{attribute 'enable_dynamic_creation'}
{attribute 'no_assign'}
FUNCTION_BLOCK FB_Stack EXTENDS FB_Collection IMPLEMENTS I_Stack
VAR_INPUT
	ipList : I_List; // List to perform operations on.
END_VAR
VAR_OUTPUT
END_VAR

(* Number of elements in the stack *)
PROPERTY _Count : T_Capacity
GET
IF THIS^.NullReferenceException() THEN _Count := -1; RETURN; END_IF
_Count := THIS^.ipList._Count;
END_GET
END_PROPERTY

PROPERTY _Error_Status : ST_ERROR
GET
IF THIS^.NullReferenceException() THEN _Error_Status := THIS^.stError; RETURN; END_IF
THIS^.stError := THIS^.ipList._Error_Status;
_Error_Status := F_Error(THIS^.stError.bSTATUS, THIS^.stError.nCODE, THIS^.stError.sSOURCE);
END_GET
END_PROPERTY

(* Checks of stack is empty.*)
PROPERTY _Is_Empty : BOOL
GET
IF THIS^.NullReferenceException() THEN _Is_Empty := TRUE; RETURN; END_IF
_Is_Empty := THIS^.ipList._Is_Empty;
END_GET
END_PROPERTY

METHOD PROTECTED CatchError : BOOL
VAR_INPUT
END_VAR
stError := THIS^.ipList._Error_Status;
CatchError := stError.bSTATUS;
END_METHOD

(* Empties/Clears/Deletes every item on the stack*)
METHOD Clear
VAR_INPUT
END_VAR
IF THIS^.NullReferenceException() THEN RETURN; END_IF
THIS^.ipList.Clear();
END_METHOD

METHOD PROTECTED NullReferenceException : BOOL
NullReferenceException := THIS^.ipList = 0;
IF NOT NullReferenceException THEN RETURN; END_IF
THIS^.RaiseException(2000+GVL_CmpErrors.ERR_INVALID_REFERENCE, 'Null or Invalid Reference');
END_METHOD

(* Get item from stack without removing it. *)
METHOD Peek : I_Stack
VAR_INPUT
	Item 	: ANY; (* Variable to store returned item value *)
	nIndex 	: DINT; (* Location of item*)
END_VAR
VAR_OUTPUT
	bSuccess : BOOL;
END_VAR
Peek := THIS^;
IF THIS^.NullReferenceException() THEN RETURN; END_IF
THIS^.ipList.Get(Item, nIndex, bSuccess => bSuccess);
END_METHOD

(* Gets and deletes item at the top of the stack *)
METHOD Pop : I_Stack
VAR_INPUT
	Item : ANY; (* Variable to store returned item value *)
END_VAR
VAR_OUTPUT
	bSuccess : BOOL;
END_VAR
VAR
	bA, bB 	 : BOOL;
END_VAR
Pop := THIS^;
IF THIS^.NullReferenceException() THEN RETURN; END_IF
THIS^.ipList.Get_First(Item, bSuccess => bA).Remove( bSuccess => bB);
bSuccess := bA AND bB;
END_METHOD

(* Removes item at the top of the stack without returning anything *)
METHOD Pop_Void : I_Stack
VAR_OUTPUT
	bSuccess : BOOL;
END_VAR
Pop_Void := THIS^;
IF THIS^.NullReferenceException() THEN RETURN; END_IF
THIS^.ipList.Remove(bSuccess => bSuccess);
END_METHOD

(* Add item to the top of the stack *)
METHOD Push : I_Stack
VAR_INPUT
	Item : ANY; (* Variable containg data to store on the stack *)
END_VAR
VAR_OUTPUT
	bSuccess : BOOL;
END_VAR
Push := THIS^;
IF THIS^.NullReferenceException() THEN RETURN; END_IF
THIS^.ipList.Add_Front(Item, bSuccess => bSuccess);
END_METHOD

(* Reverses order of items on stack *)
METHOD Reverse : I_Stack
VAR_OUTPUT
	bSuccess : BOOL;
END_VAR
Reverse := THIS^;
IF THIS^.NullReferenceException() THEN RETURN; END_IF
THIS^.ipList.Reverse(bSuccess => bSuccess);
END_METHOD

(* Get item at the top of the stack without removing it. *)
METHOD Top : I_Stack
VAR_INPUT
	Item 	: ANY; (* Variable to store returned item value *)
END_VAR
VAR_OUTPUT
	bSuccess : BOOL;
END_VAR
Top := THIS^;
IF THIS^.NullReferenceException() THEN RETURN; END_IF
THIS^.ipList.Get_First(Item, bSuccess => bSuccess);
END_METHOD

END_FUNCTION_BLOCK

(* stored: Version 1.1.0.1, ProductVersion 3.1.4024.4
   POU FB_Stack: Id {33f13e36-9900-42f1-bbaa-06171dd380dc}, SpecialFunc None
   Folder Exceptions: Id {8c4d617d-497b-4248-a944-b3a41ba5f0be}
   Folder Protected: Id {3208e573-a6ba-4628-ba51-def5ab5ae266}
   Property _Count: Id {6c6d10a0-21f3-4bac-8a60-85e10ab31bd4}
   Get Get: Id {2f584baf-f990-4f7f-93aa-d61bdaaaa2a6}
   Property _Error_Status: Id {ce73d1ee-533c-4d6a-b316-67764598fa80}
   Get Get: Id {239acf3b-26c5-40d6-ae06-2c38dc30313c}
   Property _Is_Empty: Id {c4bbeb7d-fae9-42a1-b2a4-5741ec24557f}
   Get Get: Id {4612090c-cf1a-4838-88d6-0b3ee7013bfd}
   Method CatchError: Id {0532b148-4715-4b7e-8183-5316fd5e6f33}
   Method Clear: Id {65bd9818-53a0-463c-b8c9-56e30725b5f8}
   Method NullReferenceException: Id {19bf9596-ce9c-46ad-8ef8-f87cfba22c2c}
   Method Peek: Id {1f724740-b293-42b6-af19-3d12e5260d01}
   Method Pop: Id {7d2c9231-7418-4d01-a950-6dddff60807b}
   Method Pop_Void: Id {c9348d36-9274-4a3a-ab38-d78573b18931}
   Method Push: Id {cb7bde85-03c7-45e8-8fe5-d7ebdc1b671d}
   Method Reverse: Id {ba9ac5a5-fcd7-4b04-b30f-42da8bbcce9b}
   Method Top: Id {7d111dc0-613d-4f39-bd9f-26a418db706e} *)
